TYPE TcoDiConfig :
STRUCT
    IsFalseTimeOut : TIME := T#10S;
    IsTrueTimeOut : TIME := T#10S;
END_STRUCT
END_TYPE

(* stored: Version 1.1.0.1, ProductVersion 3.1.4024.13
   DUT TcoDiConfig: Id {f20e0525-c8ac-0a6e-0986-697ac4cb18f6} *)
